(* CODESYS project Singleton_Application.project

Project tree, tasks and I/O mapping:
  Device : CODESYS Control for Raspberry Pi SL, 3S - Smart Software Solutions GmbH, version 3.5.9.40
    application Application
      libraries: Standard, * (System)
      task MainTask (cyclic, interval t#10ms, priority 1) calls PLC_PRG
      task VISU_TASK (cyclic, interval 100 ms, priority 31) calls VisuElems.Visu_Prg
      program PLC_PRG [ST]
      function block RealSingleton [ST]: fb_init, Set_Background
      global variables GVL
      function block ProxyToSingleton [ST]: fb_init, Set_Background
      interface Proxy_Interface: Set_Background
      visualisation Visualization
    SoftMotion General Axis Pool
    GPIOs_A_B : GPIOs A/B, 3S - Smart Software Solutions GmbH, version 1.1.1.10
        unmapped channels: digital inputs (GPIO0..GPIO31), digital outputs (GPIO0..GPIO31)
    I²C
    SPI
    Onewire
    Camera device
      <Empty>
  libraries: VisuSymbols, 3.5.10.0 (System)
  text list GlobalTextList
  text list System
*)

// Device/Application/GVL
{attribute 'qualified_only'}
VAR_GLOBAL CONSTANT

END_VAR

// Device/Application/PLC_PRG
PROGRAM PLC_PRG
VAR
	
	//Local possible values for background colour	
	dwBlue: DWORD := 16#FF0000FF; //Blue, highly opaque
	dwGreen: DWORD := 16#FF00FF00; //Green, highly opaque
	dwYellow: DWORD := 16#FFFFFF00; //Yellow, highly opaque

	//Creates 3 instances of the ProxyToSingleton class
	instance1	: ProxyToSingleton;
	instance2	: ProxyToSingleton;
	instance3	: ProxyToSingleton;

END_VAR

//The PLC_PRG handles the instanciation of the possible background colours and the ProxyToSingleton instances in order to be used by the Visualization element.
//The viasualization element (The client) handles the request for background change on the RealSingleton object through the ProxyToSinlgeton instances.
//These request are first processed by the ProxyToSingleton object and then passed to the one and only RealSingleton instance.
//The default background colour of the RealSingleton object is 'Blue'

END_PROGRAM

// Device/Application/ProxyToSingleton
{attribute 'enable_dynamic_creation'}
//This class is called ProxyToSingleton because it works as a Proxy of the Singleton class. It handles the creation and instanciation of the 
// RealSingleton class. Something like the proper static method GetInstance(); in any singleton pattern.
//So the ProxyToSingleton class has a static Singleton object as a field and whenever we instanciate a 
// ProxyToSingleton object we will have the RealSingleton object as its static field .realSingleton^
FUNCTION_BLOCK ProxyToSingleton IMPLEMENTS Proxy_Interface
VAR_INPUT
END_VAR
VAR_OUTPUT
END_VAR
VAR
END_VAR
VAR_STAT
		//Boolean value to check if there is already a Singleton instance
	bFirstInstance : BOOL := FALSE;
	
	//Pointer to the first and only instance of the Singleton class
	realSingleton : POINTER TO RealSingleton;
END_VAR

METHOD fb_init
VAR_INPUT
	//Needed values for instanciation.
	bInitRetains : BOOL; // TRUE: the Retain-variables are initialized (reset warm / reset cold)
 	bInCopyCode : BOOL;  // TRUE  the instance will be copied to the copy-code afterward (online change)
END_VAR
//THIS FUNCTION WORKS AS THE CONSTRUCTOR OF THE ProxyToSingleton CLASS
// It handles the creation of the only RealSingleton object. It uses the concept of lazy instanciation.

//If the static property .bFirstInstance is TRUE
IF THIS^.bFirstInstance = TRUE
	
THEN
		//There is already a Singleton object.
		//So we don't have to do anything, this new ProxyToSingleton object will already have the address of the 
		// RealSingleton object in its pointer .realSingleton
	
	ELSE	//If the static property .bFirstInstance is FALSE
	
		//There is not a Singleton object so the ProxyToSingleton object calling the constructor 
		// should create the RealSingleton object in its pointer field .realSingleton 
		//Then we change the status of the static variable bFirstInstance to TRUE and avoid overwriting the realSingleton address.
		//If the Singleton object is destroyed, .bFirstInstance should be set to FALSE again.
		THIS^.bFirstInstance := TRUE;
		
		//Reference the value of the first RealSingleton instance to the FakeSingleton object to save 
		// the address of the real Singleton instance.
		THIS^.realSingleton := __NEW(RealSingleton);
END_IF
END_METHOD

//Illustrative method of the pattern
METHOD Set_Background
VAR_INPUT
	//HEX value to be set as background color
	newBackground :DWORD;
END_VAR
//The ProxyToSingleton object handles the request and send the appropiate reques to the one and only RealSingleton instance
THIS^.realSingleton^.Set_Background(newBackground);
END_METHOD

END_FUNCTION_BLOCK

// Device/Application/RealSingleton
{attribute 'enable_dynamic_creation'}
//This class is called RealSingleton because it works as singleton.  
//As long as we only instanciate ProxyToSingleton objects, this class will work as a Singleton class should work.
//The global access point to this class is the field .realSingleton^ in every ProxyToSingleton object.

FUNCTION_BLOCK RealSingleton IMPLEMENTS Proxy_Interface
VAR_STAT
END_VAR
VAR
	//Illustrative field of the pattern to store the HEX value for the background colour
	backgroundColour : DWORD;
END_VAR

METHOD fb_init
VAR_INPUT
	//Needed values for instanciation.
	bInitRetains : BOOL; // TRUE: the Retain-variables are initialized (reset warm / reset cold)
 	bInCopyCode : BOOL;  // TRUE  the instance will be copied to the copy-code afterward (online change)
END_VAR
//The default valur for the background is set
THIS^.Set_Background(PLC_PRG.dwBlue);
END_METHOD

//Illustrative method of the pattern
METHOD Set_Background
VAR_INPUT
	//HEX value to be set as background color
	newBackground :DWORD;
END_VAR
//Writes the backgroundColour field to the passed newBackground value
THIS^.backgroundColour := newBackground;
END_METHOD

END_FUNCTION_BLOCK

// Device/Application/Proxy_Interface
INTERFACE Proxy_Interface

//Illustrative method of the pattern
METHOD Set_Background
VAR_INPUT
	//HEX value to be set as background color
	newBackground :DWORD;
END_VAR
END_METHOD

END_INTERFACE

// Device/Application/Visualization
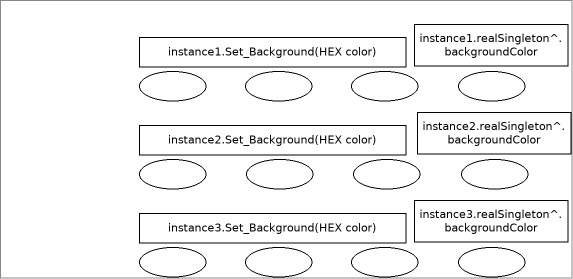
VISUALIZATION Visualization  // 573x279
//The PLC_PRG handles the instanciation of the possible background colours and the ProxyToSingleton instances in order to be used by the Visualization element.
//The viasualization element (The client) handles the request for background change on the RealSingleton object through the ProxyToSinlgeton instances.
//These request are first processed by the ProxyToSingleton object and then passed to the one and only RealSingleton instance.
//The default background colour of the RealSingleton object is 'Blue'
    Ellipse (139,71 67x30), colour variable: PLC_PRG.dwBlue
        OnMouseClick: execute { PLC_PRG.instance1.Set_Background(PLC_PRG.dwBlue); }
    Ellipse (245,71 67x30), colour variable: PLC_PRG.dwGreen
        OnMouseClick: execute { PLC_PRG.instance1.Set_Background(PLC_PRG.dwGreen); }
    Ellipse (351,71 67x30), colour variable: PLC_PRG.dwYellow
        OnMouseClick: execute { PLC_PRG.instance1.Set_Background(PLC_PRG.dwYellow); }
    Ellipse (458,71 67x30), colour variable: PLC_PRG.instance1.realSingleton^.backgroundColour
    RoundedRectangle (139,37 267x30), "instance1.Set_Background(HEX color)"
    RoundedRectangle (414,24 154x42), "instance1.realSingleton^. backgroundColor"
    Ellipse (139,159 67x30), colour variable: PLC_PRG.dwBlue
        OnMouseClick: execute { PLC_PRG.instance2.Set_Background(PLC_PRG.dwBlue); }
    Ellipse (246,159 67x30), colour variable: PLC_PRG.dwGreen
        OnMouseClick: execute { PLC_PRG.instance2.Set_Background(PLC_PRG.dwGreen); }
    Ellipse (353,159 67x30), colour variable: PLC_PRG.dwYellow
        OnMouseClick: execute { PLC_PRG.instance2.Set_Background(PLC_PRG.dwYellow); }
    Ellipse (461,159 67x30), colour variable: PLC_PRG.instance2.realSingleton^.backgroundColour
    RoundedRectangle (139,125 267x30), "instance2.Set_Background(HEX color)"
    RoundedRectangle (417,112 154x42), "instance2.realSingleton^. backgroundColor"
    Ellipse (139,247 67x30), colour variable: PLC_PRG.dwBlue
        OnMouseClick: execute { PLC_PRG.instance3.Set_Background(PLC_PRG.dwBlue); }
    Ellipse (245,247 67x30), colour variable: PLC_PRG.dwGreen
        OnMouseClick: execute { PLC_PRG.instance3.Set_Background(PLC_PRG.dwGreen); }
    Ellipse (351,247 67x30), colour variable: PLC_PRG.dwYellow
        OnMouseClick: execute { PLC_PRG.instance3.Set_Background(PLC_PRG.dwYellow); }
    Ellipse (458,247 67x30), colour variable: PLC_PRG.instance3.realSingleton^.backgroundColour
    RoundedRectangle (139,213 267x30), "instance3.Set_Background(HEX color)"
    RoundedRectangle (414,200 154x42), "instance3.realSingleton^. backgroundColor"
END_VISUALIZATION

(* text list System (id | default)
  Apr | Apr
  April | April
  Aug | Aug
  August | August
  Dec | Dec
  December | December
  Feb | Feb
  February | February
  Fri | Fri
  Friday | Friday
  Jan | Jan
  January | January
  Jul | Jul
  July | July
  Jun | Jun
  June | June
  Mar | Mar
  March | March
  May | May
  May_3Letter | May
  Mon | Mon
  Monday | Monday
  Nov | Nov
  November | November
  Oct | Oct
  October | October
  Sat | Sat
  Saturday | Saturday
  Sep | Sep
  September | September
  Sun | Sun
  Sunday | Sunday
  Thu | Thu
  Thursday | Thursday
  Tue | Tue
  Tuesday | Tuesday
  Wed | Wed
  Wednesday | Wednesday
   |  *)
